(* IEC 61131-3 sources: volt/packages/volt-lsp-iec/test-corpus/pro2193/Device/Plc Logic/Application/09 Misc/Library Manager/L_SSYP_CmpLenzeIPCSystem, 22 files *)

(* ---- L_SSYP_EVTPARAM_CMPLENZEIPCSYSTEMCAMFILECHANGED.dut ---- *)
TYPE L_SSYP_EVTPARAM_CMPLENZEIPCSYSTEMCAMFILECHANGED :
STRUCT
	STRFILENAME : STRING;
END_STRUCT
END_TYPE

(* ---- L_SSYP_EVTPARAM_CMPLENZEIPCSYSTEMSOFTPLCPARACHANGED.dut ---- *)
TYPE L_SSYP_EVTPARAM_CMPLENZEIPCSYSTEMSOFTPLCPARACHANGED :
STRUCT
	NBASEINDEX : DINT;
	NINDEX : DINT;
	BYSUBINDEX : BYTE;
END_STRUCT
END_TYPE

(* ---- L_SSYP_PERSISTANTDATAMEMORYAREA.dut ---- *)
TYPE L_SSYP_PERSISTANTDATAMEMORYAREA :
STRUCT
	PADDRESS0 : POINTER TO DWORD;
	PADDRESS1 : POINTER TO DWORD;
	PMEMVALIDFLAG : POINTER TO BOOL;
	DWSIZE : DWORD;
END_STRUCT
END_TYPE

(* ---- EVENTIDS.gvl ---- *)
VAR_GLOBAL
	CMPID_CMPLENZEIPCSYSTEM : DWORD := 16#2003;
	EVT_CMPLENZEIPCSYSTEMSOFTPLCPARACHANGED : DWORD := 16#10000009;
	EVTPARAMID_CMPLENZEIPCSYSTEMSOFTPLCPARACHANGED : WORD := 16#2;
	EVTVERSION_CMPLENZEIPCSYSTEMSOFTPLCPARACHANGED : WORD := 16#1;
	EVT_CMPLENZEIPCSYSTEMCAMFILECHANGED : DWORD := 16#1000000A;
	EVTPARAMID_CMPLENZEIPCSYSTEMCAMFILECHANGED : WORD := 16#3;
	EVTVERSION_CMPLENZEIPCSYSTEMCAMFILECHANGED : WORD := 16#1;
	EVT_CMPLENZEIPCSYSTEMPLCPARAMDESCLOADED : DWORD := 16#1000000C;
	EVTPARAMID_CMPLENZEIPCSYSTEMPLCPARAMDESCLOADED : WORD := 16#5;
	EVTVERSION_CMPLENZEIPCSYSTEMPLCPARAMDESCLOADED : WORD := 16#1;
END_VAR

(* ---- GETBOOLEANPROPERTY.pou ---- *)
FUNCTION GETBOOLEANPROPERTY : BOOL
VAR_INPUT
	STKEY : WSTRING;
END_VAR
END_FUNCTION

(* ---- GETCOMPANY.pou ---- *)
FUNCTION GETCOMPANY : WSTRING
END_FUNCTION

(* ---- GETNUMBERPROPERTY.pou ---- *)
FUNCTION GETNUMBERPROPERTY : DINT
VAR_INPUT
	STKEY : WSTRING;
END_VAR
END_FUNCTION

(* ---- GETTEXTPROPERTY.pou ---- *)
FUNCTION GETTEXTPROPERTY : WSTRING
VAR_INPUT
	STKEY : WSTRING;
END_VAR
END_FUNCTION

(* ---- GETTEXTPROPERTY2.pou ---- *)
FUNCTION GETTEXTPROPERTY2 : POINTER TO WSTRING
VAR_INPUT
	STKEY : WSTRING;
END_VAR
END_FUNCTION

(* ---- GETTITLE.pou ---- *)
FUNCTION GETTITLE : WSTRING
END_FUNCTION

(* ---- GETVERSION.pou ---- *)
FUNCTION GETVERSION : VERSION
END_FUNCTION

(* ---- GETVERSIONPROPERTY.pou ---- *)
FUNCTION GETVERSIONPROPERTY : VERSION
VAR_INPUT
	STKEY : WSTRING;
END_VAR
END_FUNCTION

(* ---- L_SSYP_DUALUSELICENSEAVAILABLE.pou ---- *)
FUNCTION L_SSYP_DUALUSELICENSEAVAILABLE : BOOL
END_FUNCTION

(* ---- L_SSYP_FORCECMEXIT.pou ---- *)
FUNCTION L_SSYP_FORCECMEXIT : BOOL
END_FUNCTION

(* ---- L_SSYP_GETPERSISTENTDATAMEMORY.pou ---- *)
FUNCTION L_SSYP_GETPERSISTENTDATAMEMORY : L_SSYP_PersistantDataMemoryArea
END_FUNCTION

(* ---- L_SSYP_GETSYSTEMTIMESTAMP.pou ---- *)
FUNCTION L_SSYP_GETSYSTEMTIMESTAMP : ULINT
VAR_INPUT
	HTASK : RTS_IEC_HANDLE;
END_VAR
END_FUNCTION

(* ---- L_SSYP_GETTASKSCHEDULERCOUNTER.pou ---- *)
FUNCTION L_SSYP_GETTASKSCHEDULERCOUNTER : DWORD
END_FUNCTION

(* ---- L_SSYP_RESETTASKSCHEDULERCOUNTER.pou ---- *)
FUNCTION L_SSYP_RESETTASKSCHEDULERCOUNTER : BOOL
END_FUNCTION

(* ---- L_SSYP_RESTOREPERSISTENTMOTIONDATA.pou ---- *)
FUNCTION L_SSYP_RESTOREPERSISTENTMOTIONDATA : RTS_IEC_RESULT
END_FUNCTION

(* ---- L_SSYP_SETBINDTODEVICE.pou ---- *)
FUNCTION L_SSYP_SETBINDTODEVICE : RTS_IEC_RESULT
VAR_INPUT
	HSOCKET : RTS_IEC_HANDLE;
	POPTIONVALUE : POINTER TO BYTE;
	DIOPTIONLEN : DINT;
END_VAR
END_FUNCTION

(* ---- L_SSYP_SIMULATIONMODEENABLED.pou ---- *)
FUNCTION L_SSYP_SIMULATIONMODEENABLED : BOOL
END_FUNCTION

(* ---- L_SSYP_STOREPERSISTENTMOTIONDATA.pou ---- *)
FUNCTION L_SSYP_STOREPERSISTENTMOTIONDATA : RTS_IEC_RESULT
END_FUNCTION
